TYPE AX5000_P_0801 :
STRUCT
	Digital_inputs_state:UINT;
END_STRUCT
END_TYPE

(* stored: Version 1.1.0.1, ProductVersion 3.1.4024.3
   DUT AX5000_P_0801: Id {3c8ee299-6a8f-4d07-880d-62ff95317902} *)
